PROGRAM MAIN
VAR
	count 				: INT := 0;
	i_CounterFun 		: INT := 0;
	i_CounterFunBlock	: INT := 0;
	i_CounterProgram	: INT := 0;
	
	fb_Count_obj1 		: Fb_Counter;
END_VAR

// count := count + 1;

// count up with counter function
i_CounterFun := Fun_Counter(i_CounterFun); 



// count up with counter function block
fb_Count_obj1();   // call function block
i_CounterFunBlock := fb_Count_obj1.i_countOut;   // access variables



// count up using a program
Prg_Counter(i_countOut => i_CounterProgram);


// access global variable list
GVL_IO.input1;

END_PROGRAM

(* stored: Version 1.1.0.1, ProductVersion 3.1.4024.9
   POU MAIN: Id {260d71a0-0831-43e2-af30-09a834cbf7a1}, SpecialFunc None *)
